{attribute 'qualified_only'}
{attribute 'strict'}
{attribute 'to_string'}
TYPE E_PackMLMode :
(
	Unknown := 0,
	Manual,
	Production
)UINT;
END_TYPE

(* stored: Version 1.1.0.1, ProductVersion 3.1.4026.18
   DUT E_PackMLMode: Id {f796ee0c-cefa-4ab5-8115-2e642d11ae3f} *)
